FUNCTION F_CoolTank : BOOL
VAR_INPUT
    refTank : REFERENCE TO ST_Tank;    
END_VAR

IF refTank.rtemperature > GVL_TankConstants.rTEMP_MIN THEN 
	refTank.rtemperature := refTank.rtemperature - GVL_TankConstants.rCOOL_RATE;
		
		IF refTank.rtemperature < GVL_TankConstants.rTEMP_MIN THEN
			refTank.rtemperature :=  GVL_TankConstants.rTEMP_MIN;
		END_IF
		
	F_CoolTank := TRUE;
ELSE
	F_CoolTank := FALSE;
END_IF

END_FUNCTION

(* stored: Version 1.1.0.1, ProductVersion 3.1.4024.16
   POU F_CoolTank: Id {23eb2f19-1862-4331-a502-53c245c36ec3}, SpecialFunc None *)
